{attribute 'qualified_only'}
{attribute 'strict'}
TYPE E_SeqLoader :
(
  cIdle           := 0,
  cStartExtend       ,
  cMovingExtend      ,
  cTargetReached      ,
  cStartRetract      ,
  cMovingRetract     ,
  cEndMovement        ,
  cError
);
END_TYPE

(* stored: Version 1.1.0.1, ProductVersion 3.1.4024.12
   DUT E_SeqLoader: Id {b4d32e7b-70e9-450c-8f06-6fa593492a50} *)
